// TIA Portal V20 export
VAR_GLOBAL   // PLC tag table "tet111"
END_VAR
